FUNCTION_BLOCK T_ComponentsCollection IMPLEMENTS I_ComponentsCollection
VAR
  _list : ARRAY[1.._collectionSize] OF I_ComponentBase;
  _collectionSize : UINT;
  _count : UINT;
END_VAR

METHOD PUBLIC AddComponent : BOOL
VAR_INPUT
  newComponent : I_ComponentBase;
END_VAR
END_METHOD

METHOD PUBLIC ContainsComponent : BOOL
VAR_INPUT
  newComponent : I_ComponentBase;
END_VAR
END_METHOD

{warning 'add property implementation'}
PROPERTY Count : UINT
GET
Count := _count;
END_GET
END_PROPERTY

{warning 'add method implementation '}
METHOD CyclicLogic
END_METHOD

METHOD FB_init : BOOL
VAR_INPUT
	bInitRetains : BOOL; // if TRUE, the retain variables are initialized (warm start / cold start)
	bInCopyCode : BOOL;  // if TRUE, the instance afterwards gets moved into the copy code (online change)
  size : UINT;
END_VAR
_collectionSize := size;
END_METHOD

METHOD PUBLIC GetComponent : BOOL
VAR_INPUT
  index : UDINT;
END_VAR
END_METHOD

{warning 'add method implementation '}
METHOD Initialize
END_METHOD

METHOD PUBLIC RemoveComponent : BOOL
VAR_INPUT
  newComponent : I_ComponentBase;
END_VAR
END_METHOD

METHOD PUBLIC RemoveComponentAt : BOOL
VAR_INPUT
  index : UDINT;
END_VAR
END_METHOD

END_FUNCTION_BLOCK

(* stored: Version 1.1.0.1, ProductVersion 3.1.4024.12
   POU T_ComponentsCollection: Id {1907c29b-927e-4ee6-99fd-d1c9ebb9baa8}, SpecialFunc None
   Method AddComponent: Id {2212367a-2ccb-4213-b9ad-535f23d61e86}
   Method ContainsComponent: Id {693bb628-e29c-4167-afa4-8c80dd6c1511}
   Property Count: Id {55e1477c-3136-4a7e-a3e4-3fe63d7e7de9}
   Get Get: Id {57426790-7eeb-497a-9a8c-3e3f26980ab3}
   Method CyclicLogic: Id {6b022d9a-6f0b-44a5-a44b-47a525b5b262}
   Method FB_init: Id {caf98cd9-019c-48a6-b62d-54994e1f37d3}
   Method GetComponent: Id {b70b2547-53b4-4a2a-86a8-7473df8a8e2e}
   Method Initialize: Id {ff827305-8660-41df-b0d9-35cc9dea669b}
   Method RemoveComponent: Id {3faecaff-22aa-4629-864d-72a7739e9361}
   Method RemoveComponentAt: Id {8292d648-1fe8-42e8-89ed-12855c33efd2} *)
